PROGRAM MAIN
VAR
END_VAR

END_PROGRAM

(* stored: Version 1.1.0.1
   POU MAIN: Id {2c15b3a3-9bd1-4015-8746-2bb1a43ab35e} *)
